(* CODESYS project helperfunctions.library
   Author: vscottki
   Placeholder: HelperFunctions
   Title: HelperFunctions
   Version: 1.0.2.0
   DocFormat: reStructuredText
   Company: Amazon

Project tree, tasks and I/O mapping:
  libraries: Tc2_Standard, * (Beckhoff Automation GmbH); Tc2_System, * (Beckhoff Automation GmbH); Tc2_Utilities, * (Beckhoff Automation GmbH); Tc3_Module, * (Beckhoff Automation GmbH)
  DUTs/
  GVLs/
    global variables GC
    global variables Param_HelperFunctions
  POUs/
    function DateTimeAsT_MaxString [ST]
    function F_MapInt [ST]
    function F_MapLReal [ST]
    function block FB_Debounce [ST]
    program MAIN [ST]
    function ReplaceInString [ST]
    function SystemTimeUtcCorrected [ST]
  Project Information/
    function F_GetCompany [ST]
    function F_GetTitle [ST]
    function F_GetVersion [ST]
  Version/
    global variables Global_Version
  VISUs/
*)

// GVLs/GC
{attribute 'qualified_only'}
VAR_GLOBAL CONSTANT
  CountOf100NsIncrement1Hr  : LINT  := 36000000000;  // do not edit  
END_VAR

// GVLs/Param_HelperFunctions
{attribute 'qualified_only'}
VAR_GLOBAL CONSTANT
  HourDeltaFromUtc          : SINT  := -7;
END_VAR

// Version/Global_Version
{attribute 'TcGenerated'}
{attribute 'no-analysis'}
{attribute 'linkalways'}
// This function has been automatically generated from the project information.
VAR_GLOBAL CONSTANT
	{attribute 'const_non_replaced'}
	stLibVersion_HelperFunctions : ST_LibVersion := (iMajor := 1, iMinor := 0, iBuild := 2, iRevision := 0, nFlags := 1, sVersion := '1.0.2.0');
END_VAR

// POUs/DateTimeAsT_MaxString
FUNCTION DateTimeAsT_MaxString : Tc2_System.T_MaxString
VAR_INPUT
  HourDeltaUTC              : SINT  := Param_HelperFunctions.HourDeltaFromUtc;
END_VAR
VAR
  timeAsFileTime            : Tc2_Utilities.T_FILETIME64;
  timeAsDt                  : DT;
  tempDtForUtcCalc          : Tc2_Utilities.T_FILETIME64;
END_VAR
VAR CONSTANT
  CountOf100NsIncrement1Hr  : LINT  := 36000000000;
END_VAR

timeAsFileTime    := Tc2_System.F_GetSystemTime();

tempDtForUtcCalc  := timeAsFileTime + (HourDeltaUTC * GC.CountOf100NsIncrement1Hr);
timeAsDt          := Tc2_Utilities.FILETIME64_TO_DT(fileTime := tempDtForUtcCalc);

DateTimeAsT_MaxString := DT_TO_STRING(timeAsDt);

END_FUNCTION

// POUs/F_MapInt
FUNCTION F_MapInt : INT
VAR_INPUT
	x : INT;
	in_min : REAL;
	in_max : REAL;
	out_min : REAL;
	out_max : REAL;
END_VAR

IF (in_max - in_min) <> 0 THEN
	F_MapInt := REAL_TO_INT((((x - in_min) * (out_max - out_min)) / (in_max - in_min)) + out_min);
ELSE
	F_MapInt := 0;
END_IF

END_FUNCTION

// POUs/F_MapLReal
FUNCTION F_MapLReal : LREAL
VAR_INPUT
	x : LREAL;
	in_min : LREAL;
	in_max : LREAL;
	out_min : LREAL;
	out_max : LREAL;
END_VAR

IF (in_max - in_min) <> 0 THEN
	F_MapLReal := (((x - in_min) * (out_max - out_min)) / (in_max - in_min)) + out_min;
ELSE
	F_MapLReal := 0;
END_IF

END_FUNCTION

// POUs/FB_Debounce
FUNCTION_BLOCK FB_Debounce
VAR_INPUT
	tOnDelay	: TIME;
	tOffDelay	: TIME;
	xRawSignal	: BOOL;
END_VAR
VAR_OUTPUT
	Debounced	: BOOL;
END_VAR
VAR
	TimerOn 	: Tc2_Standard.TON;
	TimerOff 	: Tc2_Standard.TOF;
	ftSignal	: Tc2_Standard.F_TRIG;
END_VAR

TimerOn(PT := tOnDelay);  //TON
TimerOff(PT := tOffDelay);  //TOF
ftSignal(CLK := xRawSignal);

TimerOn.IN := xRawSignal;
TimerOff.IN := ftSignal.Q; 

Debounced := TimerOn.Q OR TimerOff.Q;

END_FUNCTION_BLOCK

// POUs/MAIN
PROGRAM MAIN
VAR
  TestValueC  : ULINT;
  Datestring  : Tc2_System.T_MaxString;  
  trig        : BOOL;
  testString  : Tc2_System.T_MaxString := 'YourMotherIsAHampster';
  returnString  :Tc2_System.T_MaxString;
END_VAR

IF trig THEN
  trig        := FALSE;
  Datestring  := DateTimeAsT_MaxString(HourDeltaUTC := Param_HelperFunctions.HourDeltaFromUtc);
  returnString := 
    ReplaceInString(ObjectString := Datestring, StringToRemove := '-', StringToInsert := '#');
   returnString := 
    ReplaceInString(ObjectString := Datestring, StringToRemove := ':', StringToInsert := '#');   
END_IF

END_PROGRAM

// POUs/ReplaceInString
FUNCTION ReplaceInString : STRING
VAR_INPUT
  ObjectString    : STRING;
  StringToRemove  : STRING;
  StringToInsert  : STRING;
END_VAR
VAR
  tempString      : STRING;
  ReplacePosn     : INT;
END_VAR

tempString  := ObjectString;

WHILE(Tc2_Standard.FIND(STR1 := tempString, STR2 := StringToRemove) <> 0) DO
  ReplacePosn := Tc2_Standard.FIND(STR1 := tempString, STR2 := StringToRemove);
  tempString  := Tc2_Standard.REPLACE(L := Tc2_Standard.LEN(STR := StringToRemove), P := ReplacePosn,
                                      STR1 := tempString, STR2 := StringToInsert);
END_WHILE

ReplaceInString   := tempString;

END_FUNCTION

// POUs/SystemTimeUtcCorrected
FUNCTION SystemTimeUtcCorrected : ULINT
VAR_INPUT
  HourDeltaUTC              : SINT  := Param_HelperFunctions.HourDeltaFromUtc;
END_VAR
VAR
  timeAsFileTime            : Tc2_Utilities.T_FILETIME64;
  tempDtForUtcCalc          : Tc2_Utilities.T_FILETIME64;
END_VAR

timeAsFileTime            := Tc2_System.F_GetSystemTime();
                          
tempDtForUtcCalc          := timeAsFileTime + (HourDeltaUTC * GC.CountOf100NsIncrement1Hr);

SystemTimeUtcCorrected    := tempDtForUtcCalc;

END_FUNCTION

// Project Information/F_GetCompany
// This function has been automatically generated from the project information.
{attribute 'signature_flag' := '1073741824'}
{attribute 'TcGenerated'}
{attribute 'no-analysis'}
FUNCTION F_GetCompany : WSTRING
VAR_INPUT
	
END_VAR

F_GetCompany := "Amazon";

END_FUNCTION

// Project Information/F_GetTitle
// This function has been automatically generated from the project information.
{attribute 'signature_flag' := '1073741824'}
{attribute 'TcGenerated'}
{attribute 'no-analysis'}
FUNCTION F_GetTitle : WSTRING
VAR_INPUT
	
END_VAR

F_GetTitle := "HelperFunctions";

END_FUNCTION

// Project Information/F_GetVersion
// This function has been automatically generated from the project information.
{attribute 'signature_flag' := '1073741824'}
{attribute 'TcGenerated'}
{attribute 'no-analysis'}
FUNCTION F_GetVersion : ST_LibVersion
VAR_INPUT
	
END_VAR

F_GetVersion.iMajor := 1;
F_GetVersion.iMinor := 0;
F_GetVersion.iBuild := 2;
F_GetVersion.iRevision := 0;
F_GetVersion.sVersion := '1.0.2.0';
F_GetVersion.nFlags := 1;

END_FUNCTION
